FUNCTION_BLOCK FB_4PortViciValve
VAR_INPUT
    iAdress : INT;
END_VAR
VAR_OUTPUT
END_VAR
VAR
    fbNporValve : FB_ViciValve;
    iNumPorts : INT := 4;

    {attribute 'pytmc' := '
        pv: iReqPos
        io: io
     '}
    iReqPos : INT;
    {attribute 'pytmc' := '
        pv: SampleNames
        io: io
     '}
    stSampleNames : ST_4PViciValveSampleNames;
END_VAR

fbNporValve(iAddress := iAdress, iNumOfPorts := iNumPorts, iReqPos := iReqPos);

END_FUNCTION_BLOCK

(* stored: Version 1.1.0.1, ProductVersion 3.1.4024.12
   POU FB_4PortViciValve: Id {35f5328b-2692-4fc5-a1f1-07aefd5e56d3}, SpecialFunc None *)
